      L     L#0;
      U     "MAL1S032Par".Par.FlagProcess.ProcessActive;
      SPBN  n609; // no addition
      SET   ;
      S     "MAL1S032Par".Par.FlagProcess.Inf21; // add heat quantity
      U     "SYS_Scan0_Tick1s"; // scan 1sec
      SPBN  E609;
      L     "MAL1S032Par".Par.ProcessValue_Real.Value05; // heat quantity in kW
      +R    ;
      T     "MAL1S032Par".Par.ProcessValue_Real.Value05;
      SPA   E609;
n609: NOP   0;
      U     "MAL1S032Par".Par.FlagProcess.Inf21; // add heat quantity
      SPBN  E609;
      R     "MAL1S032Par".Par.FlagProcess.Inf21; // add heat quantity
      L     "MAL1S032Par".Par.ProcessValue_Real.Value05;
      L     3.600000e+003;
      /R    ; // from kWs to kWh
      L     1.000000e+003;
      /R    ; // from kWh to MWh
      RND   ;
      T     "MAL1S032Par".Par.ProcessValue_Real.Value06; // result to batch potokoll
      L     0.000000e+000; // clear calculator
      T     "MAL1S032Par".Par.ProcessValue_Real.Value05;
E609: NOP   0;
NETWORK
TITLE =ASW_7000: Step loading kilning
//
      U     "MAL1S032".ToASW.InfDataReady;
      U     "MAL1S032".PCRead.Step.StWait;
      U     "MAL1S032".PCWrite.ExtFuncOn.StartLoading; // PIC command "start loading"
      S     "MAL1S032Par".Par.FlagFunction_1.StepLoading; // Step loading
      R     "MAL1S032Par".Par.FlagMachine.ImpulsNullstellung;
      R     "MAL1S032Par".Par.FlagMachine.CmdTurnRevAfterLoading;
      R     "MAL1S032Par".Par.FlagMachine.CmdTurnFwdAfterLoading;
//
      SET   ;
      R     "MAL1S032".PCWrite.ExtFuncOn.StartLoading; // PIC command "start loading"
//
      U     "MAL1S032".ToASW.InfDataReady;
      U     "MAL1S032".PCRead.Step.StActive;
      U     "MAL1S032Par".Par.FlagFunction_1.StepLoading; // Step loading
      SPB   e71;
      R     "MAL1S032Par".Par.Switches1.StaOn00; // LiftingPositionRound_1
      R     "MAL1S032Par".Par.Switches1.StaOn01; // LiftingPositionRound_2
      R     "MAL1S032Par".Par.Switches1.StaOn02; // LiftingPositionRound_3
      R     "MAL1S032Par".Par.Switches1.StaOn03; // LiftingPositionRound_4
      R     "MAL1S032Par".Par.Switches1.StaOn04; // LiftingPositionRound_5
      R     "MAL1S032Par".Par.Switches1.StaOn05; // LiftingPositionRound_6
e71:  NOP   0;
      U     "MAL1S032".ToASW.InfDataReady;
      U     "MAL1S032".PCRead.Step.StActive;
      U     "MAL1S032Par".Par.FlagFunction_1.StepLoading; // Step loading
      UN    "MAL1S032Par".Par.FlagFunction_1.FinishLoading;
      UN    "MAL1S032Par".Par.FlagFunction_1.LoadEnd;
      SPBN  E700;
      U(    ;
      U(    ;
      L     "G266M".A_3111_MXZ41MA.Ma.OutPositionAngle;
      L     3460; // 346.0°
      >=I   ;
      )     ;
      O     ;
      U(    ;
      L     "G266M".A_3111_MXZ41MA.Ma.OutCntRound;
      L     L#1;
      >=D   ;
      )     ;
      )     ;
      U     "MAL1S032Par".Par.FlagFunction_1.StepLoading;
      =     "MAL1S032Par".Par.FlagFunction_0.ReducedSpeed;
//
      L     "MAL1S032Par".RecipeHeader.Loading.LiftingPositionRound_3;
      L     20; // 20°
      -I    ;
      T     "MAL1S032Par".Par.ParIntMachine.LiftingPositionRound_4;
      L     "MAL1S032Par".RecipeHeader.Loading.LoadingLevelRound_3;
      L     "MAL1S032Par".RecipeHeader.Loading.OffsetLevelNextRound;
      +I    ;
      T     "MAL1S032Par".Par.ParIntMachine.LoadingLevelRound_4;
//
      L     "MAL1S032Par".Par.ParIntMachine.LiftingPositionRound_4;
      L     20; // 20°
      -I    ;
      T     "MAL1S032Par".Par.ParIntMachine.LiftingPositionRound_5;
      L     "MAL1S032Par".Par.ParIntMachine.LoadingLevelRound_4;
      L     "MAL1S032Par".RecipeHeader.Loading.OffsetLevelNextRound;
      +I    ;
      T     "MAL1S032Par".Par.ParIntMachine.LoadingLevelRound_5;
//
      L     "MAL1S032Par".Par.ParIntMachine.LiftingPositionRound_5;
      L     20; // 20°
      -I    ;
      T     "MAL1S032Par".Par.ParIntMachine.LiftingPositionRound_6;
      L     "MAL1S032Par".Par.ParIntMachine.LoadingLevelRound_5;
      L     "MAL1S032Par".RecipeHeader.Loading.OffsetLevelNextRound;
      +I    ;
      T     "MAL1S032Par".Par.ParIntMachine.LoadingLevelRound_6;
//
      L     3600;
      L     "G266M".A_3111_MXZ41MA.Ma.Par.ParTolPosition;
      -I    ;
      L     "G266M".A_3111_MXZ41MA.Ma.OutPositionAngle;
      <=I   ;
      SPB   E700;
//
      L     "G266M".A_3111_MXZ41MA.Ma.OutPositionAngle;
      L     0;
      <I    ;
//      <=I
      SPB   E700;
//
      L     "G266M".A_3111_MXZ41MA.Ma.OutPositionAngle;
      L     10;
      /I    ;
      T     "MAL1S032Par".Par.MachineValue.ISTWERT_FAHRANTRIEB_POSI;
//
      U     "MAL1S032Par".Par.FlagFunction_1.StepLoading; // Step loading
      FP    "MAL1S032Par".Par.Switches1.StaOn08;
      =     "MAL1S032Par".Par.Switches1.StaOn09; // scan start loading
      U     "MAL1S032Par".Par.Switches1.StaOn09; // scan start loading
      SPBN  e72;
      R     "MAL1S032Par".Par.Switches1.StaOn00; // LiftingPositionRound_1
      R     "MAL1S032Par".Par.Switches1.StaOn01; // LiftingPositionRound_2
      R     "MAL1S032Par".Par.Switches1.StaOn02; // LiftingPositionRound_3
      R     "MAL1S032Par".Par.Switches1.StaOn03; // LiftingPositionRound_4
      R     "MAL1S032Par".Par.Switches1.StaOn04; // LiftingPositionRound_5
      R     "MAL1S032Par".Par.Switches1.StaOn05; // LiftingPositionRound_6
//
e72:  NOP   0;
//
      U(    ;
      L     "G266M".A_3111_MXZ41MA.Ma.OutCntRound;
      L     L#0;
      ==D   ;
      )     ;
      U(    ;
      L     "MAL1S032Par".Par.MachineValue.ISTWERT_FAHRANTRIEB_POSI;
      L     "MAL1S032Par".RecipeHeader.Loading.LiftingPositionRound_1;
      <I    ;
      )     ;
      S     "MAL1S032Par".Par.Switches1.StaOn00; // LiftingPositionRound_1
//
      U(    ;
      L     "G266M".A_3111_MXZ41MA.Ma.OutCntRound;
      L     L#0;
      ==D   ;
      )     ;
      U(    ;
      L     "MAL1S032Par".Par.MachineValue.ISTWERT_FAHRANTRIEB_POSI;
      L     "MAL1S032Par".RecipeHeader.Loading.LiftingPositionRound_1;
      >=I   ;
      )     ;
      U(    ;
      L     "MAL1S032Par".Par.MachineValue.ISTWERT_FAHRANTRIEB_POSI;
      L     3550; // 355.0° --> Ruckeln am Nullpunkt abfangen
      <=I   ;
      )     ;
      S     "MAL1S032Par".Par.Switches1.StaOn01; // LiftingPositionRound_2
//
      U     "MAL1S032Par".Par.Switches1.StaOn01; // LiftingPositionRound_2
      R     "MAL1S032Par".Par.Switches1.StaOn00; // LiftingPositionRound_1
//
      U(    ;
      L     "G266M".A_3111_MXZ41MA.Ma.OutCntRound;
      L     L#1;
      ==D   ;
      )     ;
      U(    ;
      L     "MAL1S032Par".Par.MachineValue.ISTWERT_FAHRANTRIEB_POSI;
      L     "MAL1S032Par".RecipeHeader.Loading.LiftingPositionRound_2;
      >=I   ;
      )     ;
      S     "MAL1S032Par".Par.Switches1.StaOn02; // LiftingPositionRound_3
//
      U     "MAL1S032Par".Par.Switches1.StaOn02; // LiftingPositionRound_3
      R     "MAL1S032Par".Par.Switches1.StaOn01; // LiftingPositionRound_2
      R     "MAL1S032Par".Par.Switches1.StaOn00; // LiftingPositionRound_1
//
      U(    ;
      L     "G266M".A_3111_MXZ41MA.Ma.OutCntRound;
      L     L#2;
      ==D   ;
      )     ;
      U(    ;
      L     "MAL1S032Par".Par.MachineValue.ISTWERT_FAHRANTRIEB_POSI;
      L     "MAL1S032Par".RecipeHeader.Loading.LiftingPositionRound_3;
      >=I   ;
      )     ;
      S     "MAL1S032Par".Par.Switches1.StaOn03; // LiftingPositionRound_4
//
      U     "MAL1S032Par".Par.Switches1.StaOn03; // LiftingPositionRound_4
      R     "MAL1S032Par".Par.Switches1.StaOn02; // LiftingPositionRound_3
      R     "MAL1S032Par".Par.Switches1.StaOn01; // LiftingPositionRound_2
      R     "MAL1S032Par".Par.Switches1.StaOn00; // LiftingPositionRound_1
      U(    ;
      L     "G266M".A_3111_MXZ41MA.Ma.OutCntRound;
      L     L#3;
      ==D   ;
      )     ;
      U(    ;
      L     "MAL1S032Par".Par.MachineValue.ISTWERT_FAHRANTRIEB_POSI;
      L     "MAL1S032Par".Par.ParIntMachine.LiftingPositionRound_4;
      >=I   ;
      )     ;
      S     "MAL1S032Par".Par.Switches1.StaOn04; // LiftingPositionRound_5
//
      U     "MAL1S032Par".Par.Switches1.StaOn04; // LiftingPositionRound_5
      R     "MAL1S032Par".Par.Switches1.StaOn03; // LiftingPositionRound_4
      R     "MAL1S032Par".Par.Switches1.StaOn02; // LiftingPositionRound_3
      R     "MAL1S032Par".Par.Switches1.StaOn01; // LiftingPositionRound_2
      R     "MAL1S032Par".Par.Switches1.StaOn00; // LiftingPositionRound_1
      U(    ;
      L     "G266M".A_3111_MXZ41MA.Ma.OutCntRound;
      L     L#4;
      ==D   ;
      )     ;
      U(    ;
      L     "MAL1S032Par".Par.MachineValue.ISTWERT_FAHRANTRIEB_POSI;
      L     "MAL1S032Par".Par.ParIntMachine.LiftingPositionRound_5;
      >=I   ;
      )     ;
      S     "MAL1S032Par".Par.Switches1.StaOn05; // LiftingPositionRound_6
//
      U     "MAL1S032Par".Par.Switches1.StaOn05; // LiftingPositionRound_6
      R     "MAL1S032Par".Par.Switches1.StaOn04; // LiftingPositionRound_5
      R     "MAL1S032Par".Par.Switches1.StaOn03; // LiftingPositionRound_4
      R     "MAL1S032Par".Par.Switches1.StaOn02; // LiftingPositionRound_3
      R     "MAL1S032Par".Par.Switches1.StaOn01; // LiftingPositionRound_2
      R     "MAL1S032Par".Par.Switches1.StaOn00; // LiftingPositionRound_1
      U     "MAL1S032Par".Par.Switches1.StaOn00; // LiftingPositionRound_1
      SPB   Rnd1;
      U     "MAL1S032Par".Par.Switches1.StaOn01; // LiftingPositionRound_2
      SPB   Rnd2;
      U     "MAL1S032Par".Par.Switches1.StaOn02; // LiftingPositionRound_3
      SPB   Rnd3;
      U     "MAL1S032Par".Par.Switches1.StaOn03; // LiftingPositionRound_4
      SPB   Rnd4;
      U     "MAL1S032Par".Par.Switches1.StaOn04; // LiftingPositionRound_5
      SPB   Rnd5;
      U     "MAL1S032Par".Par.Switches1.StaOn05; // LiftingPositionRound_6
      SPB   Rnd6;
      SPA   E700;
Rnd1: NOP   0;
      L     "MAL1S032Par".RecipeHeader.Loading.LoadingLevelRound_1;
      L     "G265M".A_3111_MXZ21_31MA.Ma.Par.ParTolPosition;
      +I    ;
      T     "MAL1S032Par".Par.MachineValue.SOLLWERT_HUBZUG1_HOEHE;
      T     "MAL1S032Par".Par.MachineValue.SOLLWERT_HUBZUG2_HOEHE;
      L     "MAL1S032Par".RecipeHeader.Loading.LoadingSpeed_1;
      T     "MAL1S032Par".Par.MachineValue.SollwertFahrantrieb;
      SPA   E700;
Rnd2: NOP   0;
      L     "MAL1S032Par".RecipeHeader.Loading.LoadingLevelRound_2;
      L     "G265M".A_3111_MXZ21_31MA.Ma.Par.ParTolPosition;
      +I    ;
      T     "MAL1S032Par".Par.MachineValue.SOLLWERT_HUBZUG1_HOEHE;
      T     "MAL1S032Par".Par.MachineValue.SOLLWERT_HUBZUG2_HOEHE;
      L     "MAL1S032Par".RecipeHeader.Loading.LoadingSpeed_2;
      T     "MAL1S032Par".Par.MachineValue.SollwertFahrantrieb;
      SPA   E700;
Rnd3: NOP   0;
      L     "MAL1S032Par".RecipeHeader.Loading.LoadingLevelRound_3;
      L     "G265M".A_3111_MXZ21_31MA.Ma.Par.ParTolPosition;
      +I    ;
      T     "MAL1S032Par".Par.MachineValue.SOLLWERT_HUBZUG1_HOEHE;
      T     "MAL1S032Par".Par.MachineValue.SOLLWERT_HUBZUG2_HOEHE;
      L     "MAL1S032Par".RecipeHeader.Loading.LoadingSpeed_3;
      T     "MAL1S032Par".Par.MachineValue.SollwertFahrantrieb;
      SPA   E700;
Rnd4: NOP   0;
      L     "MAL1S032Par".Par.ParIntMachine.LoadingLevelRound_4;
      L     "G265M".A_3111_MXZ21_31MA.Ma.Par.ParTolPosition;
      +I    ;
      T     "MAL1S032Par".Par.MachineValue.SOLLWERT_HUBZUG1_HOEHE;
      T     "MAL1S032Par".Par.MachineValue.SOLLWERT_HUBZUG2_HOEHE;
//      L     "MAL1S032Par".RecipeHeader.Loading.LoadingSpeed_3
      L     87; // 87%
      T     "MAL1S032Par".Par.MachineValue.SollwertFahrantrieb;
      SPA   E700;
Rnd5: NOP   0;
      L     "MAL1S032Par".Par.ParIntMachine.LoadingLevelRound_5;
      L     "G265M".A_3111_MXZ21_31MA.Ma.Par.ParTolPosition;
      +I    ;
      T     "MAL1S032Par".Par.MachineValue.SOLLWERT_HUBZUG1_HOEHE;
      T     "MAL1S032Par".Par.MachineValue.SOLLWERT_HUBZUG2_HOEHE;
//      L     "MAL1S032Par".RecipeHeader.Loading.LoadingSpeed_3
      L     87; // 87%
      T     "MAL1S032Par".Par.MachineValue.SollwertFahrantrieb;
      SPA   E700;
Rnd6: NOP   0;
      L     "MAL1S032Par".Par.ParIntMachine.LoadingLevelRound_6;
      L     "G265M".A_3111_MXZ21_31MA.Ma.Par.ParTolPosition;
      +I    ;
      T     "MAL1S032Par".Par.MachineValue.SOLLWERT_HUBZUG1_HOEHE;
      T     "MAL1S032Par".Par.MachineValue.SOLLWERT_HUBZUG2_HOEHE;
//      L     "MAL1S032Par".RecipeHeader.Loading.LoadingSpeed_3
      L     87; // 87%
      T     "MAL1S032Par".Par.MachineValue.SollwertFahrantrieb;
      SPA   E700;
E700: NOP   0;
NETWORK
TITLE =Sub 7010: Kilning  loading finished

// Grundschicht vollständig bedeckt
      U(    ;
// Die Position bei IBN ermitteln!
      L     "G266M".A_3111_MXZ41MA.Ma.OutPositionAngle;
      L     3564; // 356.4°
      >=I   ;
      )     ;
      U     "MAL1S032Par".Par.FlagFunction_1.StepLoading;
      U     "G266M".A_3111_MXZ41MA.Ma.InEnableFwd;
      S     "MAL1S032Par".Par.FlagFunction_1.LoadFirstPartEnd;
      S     "MAL1S032Par".Par.FlagProcess.Product_Inside;

      U     "MAL1S032Par".Par.FlagProcess.ProcessActive;
      U     "MAL1S032Par".Par.FlagFunction_1.FinishLoading;
      O     "MAL1S032Par".Par.FlagFunction_1.StepUnloading;
      O     "MAL1S032".PCRead.Step.StIdling; // "SecDB".PCRead.Step.StIdling
      R     "MAL1S032Par".Par.FlagFunction_1.LoadFirstPartEnd;

      L     0;
      L     "MAL1S032".ToSSW.InPrevSecDB;
      ==I   ;
      SPB   fin;
      O(    ;
      U     "MAL1S017Par".Par.FlagFunction_1.FinishUnloading;
      U     "MAL1S017".PCWrite.ExtFuncOn.FinishCleanSurface; // PIC command "finish unloading"
//      U     "MAL1S032".PCWrite.ExtFuncOn.FinishLoading    // PIC command "finish loading"
      O     "MAL1S017Par".Par.FlagFunction_1.StepCleaning;
      U     "MAL1S017".PCRead.Step.StEmptied;
      U(    ;
      AUF   "MAL1S017";
      L     DBNO;
      L     "MAL1S032".ToSSW.InPrevSecDB;
      ==I   ;
      )     ;
      )     ;
      O(    ;
      U     "MAL1S018Par".Par.FlagFunction_1.FinishUnloading;
      U     "MAL1S018".PCWrite.ExtFuncOn.FinishCleanSurface; // PIC command "finish unloading"
//      U     "MAL1S032".PCWrite.ExtFuncOn.FinishLoading    // PIC command "finish loading"
      O     "MAL1S018Par".Par.FlagFunction_1.StepCleaning;
      U     "MAL1S018".PCRead.Step.StEmptied;
      U(    ;
      AUF   "MAL1S018";
      L     DBNO;
      L     "MAL1S032".ToSSW.InPrevSecDB;
      ==I   ;
      )     ;
      )     ;
      O(    ;
      U     "MAL1S019Par".Par.FlagFunction_1.FinishUnloading;
      U     "MAL1S019".PCWrite.ExtFuncOn.FinishCleanSurface; // PIC command "finish unloading"
//      U     "MAL1S032".PCWrite.ExtFuncOn.FinishLoading    // PIC command "finish loading"
      O     "MAL1S019Par".Par.FlagFunction_1.StepCleaning;
      U     "MAL1S019".PCRead.Step.StEmptied;
      U(    ;
      AUF   "MAL1S019";
      L     DBNO;
      L     "MAL1S032".ToSSW.InPrevSecDB;
      ==I   ;
      )     ;
      )     ;
      O(    ;
      U     "MAL1S020Par".Par.FlagFunction_1.FinishUnloading;
      U     "MAL1S020".PCWrite.ExtFuncOn.FinishCleanSurface; // PIC command "finish unloading"
//      U     "MAL1S032".PCWrite.ExtFuncOn.FinishLoading    // PIC command "finish loading"
      O     "MAL1S020Par".Par.FlagFunction_1.StepCleaning;
      U     "MAL1S020".PCRead.Step.StEmptied;
      U(    ;
      AUF   "MAL1S020";
      L     DBNO;
      L     "MAL1S032".ToSSW.InPrevSecDB;
      ==I   ;
      )     ;
      )     ;
      O(    ;
      U     "MAL1S021Par".Par.FlagFunction_1.FinishUnloading;
      U     "MAL1S021".PCWrite.ExtFuncOn.FinishCleanSurface; // PIC command "finish unloading"
//      U     "MAL1S032".PCWrite.ExtFuncOn.FinishLoading    // PIC command "finish loading"
      O     "MAL1S021Par".Par.FlagFunction_1.StepCleaning;
      U     "MAL1S021".PCRead.Step.StEmptied;
      U(    ;
      AUF   "MAL1S021";
      L     DBNO;
      L     "MAL1S032".ToSSW.InPrevSecDB;
      ==I   ;
      )     ;
      )     ;
      O(    ;
      U     "MAL1S022Par".Par.FlagFunction_1.FinishUnloading;
      U     "MAL1S022".PCWrite.ExtFuncOn.FinishCleanSurface; // PIC command "finish unloading"
//      U     "MAL1S032".PCWrite.ExtFuncOn.FinishLoading    // PIC command "finish loading"
      O     "MAL1S022Par".Par.FlagFunction_1.StepCleaning;
      U     "MAL1S022".PCRead.Step.StEmptied;
      U(    ;
      AUF   "MAL1S022";
      L     DBNO;
      L     "MAL1S032".ToSSW.InPrevSecDB;
      ==I   ;
      )     ;
      )     ;
      O(    ;
      U     "MAL1S023Par".Par.FlagFunction_1.FinishUnloading;
      U     "MAL1S023".PCWrite.ExtFuncOn.FinishCleanSurface; // PIC command "finish unloading"
//      U     "MAL1S032".PCWrite.ExtFuncOn.FinishLoading    // PIC command "finish loading"
      O     "MAL1S032Par".Par.FlagFunction_1.StepCleaning;
      U     "MAL1S032".PCRead.Step.StEmptied;
      U(    ;
      AUF   "MAL1S023";
      L     DBNO;
      L     "MAL1S023".ToSSW.InPrevSecDB;
      ==I   ;
      )     ;
      )     ;
      O(    ;
      U     "MAL1S024Par".Par.FlagFunction_1.FinishUnloading;
      U     "MAL1S024".PCWrite.ExtFuncOn.FinishCleanSurface; // PIC command "finish unloading"
//      U     "MAL1S032".PCWrite.ExtFuncOn.FinishLoading    // PIC command "finish loading"
      O     "MAL1S024Par".Par.FlagFunction_1.StepCleaning;
      U     "MAL1S024".PCRead.Step.StEmptied;
      U(    ;
      AUF   "MAL1S024";
      L     DBNO;
      L     "MAL1S032".ToSSW.InPrevSecDB;
      ==I   ;
      )     ;
      )     ;
//      O(
//      U     "MAL1S032Par".Par.FlagFunction_1.StepLoading    // Step loading
//      UN    "MAL1S032".ToASW.InfSameJobPrevSec
//      U     "MAL1S032".PCWrite.ExtFuncOn.FinishLoading    // PIC command "finish loading"
//      )
      U     "MAL1S032".ToASW.InfDataReady;
      U     "MAL1S032".PCRead.Step.StActive;
      U     "MAL1S032Par".Par.FlagFunction_1.LoadFirstPartEnd;
      S     "MAL1S032Par".Par.FlagFunction_1.LoadEnd;
      R     "MAL1S017".PCWrite.ExtFuncOn.FinishCleanSurface; // PIC command "finish unloading"
      R     "MAL1S018".PCWrite.ExtFuncOn.FinishCleanSurface; // PIC command "finish unloading"
      R     "MAL1S019".PCWrite.ExtFuncOn.FinishCleanSurface; // PIC command "finish unloading"
      R     "MAL1S020".PCWrite.ExtFuncOn.FinishCleanSurface; // PIC command "finish unloading"
      R     "MAL1S021".PCWrite.ExtFuncOn.FinishCleanSurface; // PIC command "finish unloading"
      R     "MAL1S022".PCWrite.ExtFuncOn.FinishCleanSurface; // PIC command "finish unloading"
      R     "MAL1S023".PCWrite.ExtFuncOn.FinishCleanSurface; // PIC command "finish unloading"
      R     "MAL1S024".PCWrite.ExtFuncOn.FinishCleanSurface; // PIC command "finish unloading"

//
      U     "MAL1S032".PCWrite.ExtFuncOn.FinishLoading; // PIC command "finish loading"
      R     "MAL1S032".PCWrite.ExtFuncOn.FinishLoading; // PIC command "finish loading"
//
      U     "MAL1S032Par".Par.FlagFunction_1.LoadEnd;
      U     "MAL1S032Par".Par.FlagFunction_1.StepLoading; // Step loading
      FP    "MAL1S032Par".Par.FlagFunction_0.ImpulsSollposition;
      =     "MAL1S032Par".Par.FlagFunction_0.MerkerSollpositionFP;
      U     "MAL1S032Par".Par.FlagFunction_0.MerkerSollpositionFP;
      SPBN  fin;
      L     "G266M".A_3111_MXZ41MA.Ma.OutPositionAngle;
      L     "MAL1S032Par".Par.ParIntProcess.LoadingOverlap;
      +I    ;
      T     "G266M".A_3111_MXZ41MA.Ma.InPositionTarget;
      SET   ;
      S     "G266M".TurningTo_Parkposition;

// Extra Planierrunde wenn der Fahrantrieb ueber 346° beim Beladen Ende war
      L     "G266M".A_3111_MXZ41MA.Ma.OutPositionAngle;
      L     3460; // 346,0 °
      >I    ;
      S     "G266M".Turning_One_Round_More;

// Beladehöhe speichern
      L     "MAL1S032Par".Par.MachineValue.SOLLWERT_HUBZUG1_HOEHE;
      T     "MAL1S032Par".Par.ParIntMachine.LastLoadingLevel; // saved loading value
fin:  NOP   0;

// Hubzüge erst auf der Parkposition abheben
      U     "G266M".TurningTo_Parkposition;
      FN    "G265M".USW8;
      =     "G265M".USW9;

      U     "G265M".USW9;
      O     ;
      U     "MAL1S032Par".Par.FlagFunction_1.FinishLoading;
      U(    ;
      U     "G266M".A_3111_MXZ41MA.A_3111_BZS43.StCtoTrue; // sensor zero point
      O     "G266M".A_3111_MXZ41MA.A_3111_BZS43.StTrue; // sensor zero point
      )     ;
      SPBN  auf;
      L     "G265M".A_3111_MXZ21_31MA.Ma.Par.ParPositionTopLeftUnits; //LIFTING DRIVE
      L     150;
      +I    ;
      T     "MAL1S032Par".Par.MachineValue.SOLLWERT_HUBZUG1_HOEHE;
      L     "G265M".A_3111_MXZ21_31MA.Ma.Par.ParPositionTopRightUnits; //LIFTING DRIVE
      L     150;
      +I    ;
      T     "MAL1S032Par".Par.MachineValue.SOLLWERT_HUBZUG2_HOEHE;
      L     1;
      T     "G265M".A_3111_MXZ21_31MA.Ma.Par.ParTolPosition;
auf:  NOP   0;

      NOP   0;
NETWORK
TITLE =ASW_6080: Processtime Kilning
//      CALL  "SSA_MH_ProcessTime_Fct" , DB1017
//       InfDataReady :="MAL1S017".ToASW.InfDataReady
//       ProzessActive:="MAL1S017Par".Par.FlagProcess.ProcessActive
//       InStartTime  :="MAL1S017Par".Prozesstime.Starttime
//       OutStartTime :="MAL1S017Par".Prozesstime.Starttime
//       ProcessTime  :="MAL1S017Par".Prozesstime
//
      CALL "SSA_MH_ProcessTime_Fct" , DB  1032 (
           InfDataReady             := "MAL1S032".ToASW.InfDataReady,
           ProzessActive            := "MAL1S032Par".Par.FlagProcess.ProcessActive,
           InStartTime              := "MAL1S032Par".Processtime.StartTime,
           OutStartTime             := "MAL1S032Par".Processtime.StartTime,
           ProcessTime              := "MAL1S032Par".Processtime);

NETWORK
TITLE =Sub 7020: Step start process kilning

      U     "MAL1S032".ToASW.InfDataReady;
      U     "MAL1S032".PCRead.Step.StActive;
//      U     "MAL1S032".PCWrite.ExtFuncOn.StartProcess    // PIC command "start process kilning"
      U     "MAL1S032Par".Par.FlagFunction_1.LoadEnd;

      U     "G266M".A_3111_MXZ41MA.A_3111_BZS43.StTrue; // sensor zero point
      U     "G265M".A_3111_MXZ21_31MA.A_3111_BZS23.InpTrue;
      U     "G265M".A_3111_MXZ21_31MA.A_3111_BZS33.InpTrue;

      O(    ;
      UN    "MAL1S032".SecNom.Par1On.Cmd01; // With Loading
      UN    "MAL1S032".ToASW.InfSameBatchPrevSec;
      U     "MAL1S032".ToASW.InfDataReady;
      U     "MAL1S032".PCRead.Step.StActive;
      )     ;

      S     "MAL1S032Par".Par.FlagFunction_1.FinishLoading; // start process kilning
      R     "MAL1S032Par".Par.FlagFunction_1.LoadEnd;
//
      U     "MAL1S032".PCWrite.ExtFuncOn.StartProcess; // PIC command "start process kilning"
      R     "MAL1S032".PCWrite.ExtFuncOn.StartProcess; // PIC command "start process kilning"
//
      U     "G266M".A_3111_MXZ41MA.Ma.StAdjusted;
      O     "G266M".A_3111_MXZ41MA.Ma.OutAdjusted;
      U     "MAL1S032Par".Par.FlagFunction_1.FinishLoading; // start process kilning
      O     "MAL1S032Par".Par.FlagProcess.ProcessActive;
      SPBN  E702;
      L     "G265M".A_3111_MXZ21_31MA.Ma.Par.ParPositionTopLeftUnits; //LIFTING DRIVE
      L     50; //jk
      +I    ;
      T     "MAL1S032Par".Par.MachineValue.SOLLWERT_HUBZUG1_HOEHE;
      L     "G265M".A_3111_MXZ21_31MA.Ma.Par.ParPositionTopRightUnits; //LIFTING DRIVE
      L     50; //jk
      +I    ;
      T     "MAL1S032Par".Par.MachineValue.SOLLWERT_HUBZUG2_HOEHE;
      L     1;
      T     "G265M".A_3111_MXZ21_31MA.Ma.Par.ParTolPosition;

E702: NOP   0;

      U     "G266M".TurningTo_Parkposition;
      SPBN  E703;
      U(    ;
      L     "G266M".A_3111_MXZ41MA.Ma.OutPositionAngle;
      L     3500;
      >=I   ;
      )     ;
      SPBN  E703;
      L     10; // 10% speed to parkposition
      T     "MAL1S032Par".Par.MachineValue.SollwertFahrantrieb;
E703: NOP   0;

      U     "G266M".TurningTo_Parkposition;
      SPBN  E704;
      U(    ;
      L     "G266M".A_3111_MXZ41MA.Ma.OutPositionAngle;
      L     3500;
      <I    ;
      )     ;
      SPBN  E704;
      L     87; // 87% speed to parkposition
      T     "MAL1S032Par".Par.MachineValue.SollwertFahrantrieb;
E704: NOP   0;

NETWORK
TITLE =ASW_8000:  Step unloading kilning

      UN    "MAL1S032Par".Par.FlagFunction_1.StepUnloading; // Step Unloading
      R     "MAL1S032Par".Par.FlagFunction_0.OverlapSaved; // Ueberlappung erfasst
//
      U     "MAL1S032".ToASW.InfDataReady;
      U     "MAL1S032".PCRead.Step.StEmptying;
      U(    ;
      L     "MAL1S032Par".RecipeHeader.Unloading.StartUnloadAuto; //StartUnloadAuto = 0
      L     1;
      <>I   ;
      U     "MAL1S032".PCWrite.ExtFuncOn.StartUnLoading; // PIC command "start unloading"
      O     ;
      U(    ;
      L     "MAL1S032Par".RecipeHeader.Unloading.StartUnloadAuto; //StartUnloadAuto = 10
      L     1;
      ==I   ;
      )     ;
      UN    DB371.DBX  832.1; // 30% Ventilatordrehzahl
      UN    DB371.DBX 1856.1; // 30% Ventilatordrehzahl
      )     ;
      S     "MAL1S032Par".Par.FlagFunction_1.StepUnloading; // Step Unloading
      R     "MAL1S032Par".Par.FlagMachine.ImpulsNullstellung;
      R     "MAL1S023Par".Par.FlagMachine.WEGMESSUNG_0;
      R     DB922.DBX  148.0; // FP
      R     "MAL1S032Par".Par.FlagMachine.CmdTurnRevAfterUnloading;
      R     "MAL1S032Par".Par.FlagMachine.CmdTurnFwdAfterUnloading;
//
      SET   ;
      R     "MAL1S032".PCWrite.ExtFuncOn.StartUnLoading; // PIC command "start unloading"
//
      U     "MAL1S032".ToASW.InfDataReady;
      U     "MAL1S032".PCRead.Step.StEmptying;
      U     "MAL1S032Par".Par.FlagFunction_1.StepUnloading; // Step Unloading
      SPBN  e800;
      L     "MAL1S032Par".Par.ParIntMachine.LastLoadingLevel; // saved loading value
      T     "MAL1S032Par".Par.ParIntMachine.FUELLHOEHE_PRODUKT;
//
      U(    ;
      L     "G265M".A_3111_MXZ21_31MA.Ma.OutPositionLeft;
      L     "MAL1S032Par".Par.ParIntMachine.FUELLHOEHE_PRODUKT;
      >I    ;
      )     ;
      O(    ;
      L     "G265M".A_3111_MXZ21_31MA.Ma.OutPositionRight;
      L     "MAL1S032Par".Par.ParIntMachine.FUELLHOEHE_PRODUKT;
      >I    ;
      )     ;
      UN(   ;
      U(    ;
      L     "G265M".A_3111_MXZ21_31MA.Ma.OutPositionLeft;
      L     "MAL1S032Par".Par.MachineValue.SOLLWERT_HUBZUG1_HOEHE;
      <=I   ;
      )     ;
      U(    ;
      L     "G265M".A_3111_MXZ21_31MA.Ma.OutPositionRight;
      L     "MAL1S032Par".Par.MachineValue.SOLLWERT_HUBZUG1_HOEHE;
      <=I   ;
      )     ;
      )     ;
      =     "MAL1S032Par".Par.FlagFunction_0.ScrewAboveProductLayer; // HubzuegeUeberProdukt
//
//- Letzte Entladehoehe erreicht ---
      U(    ;
      L     "MAL1S032Par".Par.MachineValue.SOLLWERT_HUBZUG1_HOEHE;
      L     0;
      <=I   ;
      )     ;
      U(    ;
      L     "MAL1S032Par".Par.MachineValue.SOLLWERT_HUBZUG1_HOEHE;
      L     "G265M".A_3111_MXZ21_31MA.Ma.InPositionTarget;
      ==I   ;
      )     ;
      U     "G265M".A_3111_MXZ21_31MA.Ma.StAdjusted;
      U     "MAL1S032Par".Par.FlagFunction_1.StepUnloading; // Step Unloading
      FP    "MAL1S032Par".Par.FlagFunction_0.UnloadLevelReachedFP; // UnloadLevelReachedFP
      =     "MAL1S032Par".Par.FlagFunction_0.ImpulsUnloadLevelReached; // ImpulsUnloadLevelReached
      UN    "MAL1S032Par".Par.FlagFunction_0.ImpulsUnloadLevelReached; // ImpulsUnloadLevelReached
      O     "MAL1S032Par".Par.FlagFunction_0.OverlapSaved; // Ueberlappung erfasst
      SPB   over;
      L     "G266M".A_3111_MXZ41MA.Ma.OutCntRound;
      L     1;
      +I    ;
      T     "MAL1S032Par".Par.ParIntProcess.UnloadungRounds;
//
      L     "G266M".A_3111_MXZ41MA.Ma.OutPositionAngle;
      L     3600; // 360,0°
      >=I   ;
      SPBN  soz1;
      -I    ;
      SPA   soz2;
soz1: NOP   0;
      TAK   ;
soz2: NOP   0;
      L     100; // 10,0°
      +I    ;
      T     "MAL1S032Par".Par.ParIntProcess.UnloadingOverlap;
      T     "G266M".A_3111_MXZ41MA.Ma.InPositionTarget;
      S     "MAL1S032Par".Par.FlagFunction_0.OverlapSaved; // Ueberlappung erfasst
over: NOP   0;
      U(    ;
      L     "G266M".A_3111_MXZ41MA.Ma.OutCntRound;
      L     L#0;
      ==D   ;
      )     ;
      SPB   rnd1;
      L     "G266M".A_3111_MXZ41MA.Ma.OutCntRound;
      L     L#1;
      ==D   ;
      SPB   rnd2;
      L     "G266M".A_3111_MXZ41MA.Ma.OutCntRound;
      L     L#2;
      >=D   ;
      SPB   rnd3;
      SPA   e801;
rnd1: NOP   0;
      L     "MAL1S032Par".RecipeHeader.Unloading.UnLoadingLevelRound_1;
      T     "MAL1S032Par".Par.MachineValue.SOLLWERT_HUBZUG1_HOEHE;
      T     "MAL1S032Par".Par.MachineValue.SOLLWERT_HUBZUG2_HOEHE;
      L     1;
      T     "G265M".A_3111_MXZ21_31MA.Ma.Par.ParTolPosition;
      L     "MAL1S032Par".RecipeHeader.Unloading.UnLoadingSpeed_1;
      T     "MAL1S032Par".Par.MachineValue.SollwertFahrantrieb;
      SPA   e801;
rnd2: NOP   0;
      L     "MAL1S032Par".RecipeHeader.Unloading.UnLoadingLevelRound_2;
      T     "MAL1S032Par".Par.MachineValue.SOLLWERT_HUBZUG1_HOEHE;
      T     "MAL1S032Par".Par.MachineValue.SOLLWERT_HUBZUG2_HOEHE;
      L     1;
      T     "G265M".A_3111_MXZ21_31MA.Ma.Par.ParTolPosition;
      L     "MAL1S032Par".RecipeHeader.Unloading.UnLoadingSpeed_2;
      T     "MAL1S032Par".Par.MachineValue.SollwertFahrantrieb;
      SPA   e801;
rnd3: NOP   0;
      L     "MAL1S032Par".RecipeHeader.Unloading.UnLoadingLevelRound_3;
      T     "MAL1S032Par".Par.MachineValue.SOLLWERT_HUBZUG1_HOEHE;
      T     "MAL1S032Par".Par.MachineValue.SOLLWERT_HUBZUG2_HOEHE;
      L     1;
      T     "G265M".A_3111_MXZ21_31MA.Ma.Par.ParTolPosition;
      L     "MAL1S032Par".RecipeHeader.Unloading.UnLoadingSpeed_3;
      T     "MAL1S032Par".Par.MachineValue.SollwertFahrantrieb;
      SPA   e801;

e801: NOP   0;
      U     "MAL1S032".ToASW.InfDataReady;
      U     "MAL1S032".PCRead.Step.StEmptying;
      U     "MAL1S032Par".Par.FlagFunction_1.StepUnloading; // Step Unloading
      U(    ;
      L     "G266M".A_3111_MXZ41MA.Ma.OutCntRound;
      L     "MAL1S032Par".Par.ParIntProcess.UnloadungRounds;
      >=I   ;
      )     ;
      U     "G265M".A_3111_MXZ21_31MA.Ma.StAdjusted;
      U     "G266M".A_3111_MXZ41MA.Ma.StAdjusted;
      S     "MAL1S032Par".Par.FlagFunction_1.FinishUnloading;

      U     "MAL1S032".ToASW.InfDataReady;
      U     "MAL1S032".PCRead.Step.StEmptying;
      U     "MAL1S032Par".Par.FlagFunction_1.FinishUnloading;
      SPBN  e800;
      L     "G265M".A_3111_MXZ21_31MA.Ma.Par.ParPositionTopLeftUnits;
      L     50;
      +I    ;
      T     "MAL1S032Par".Par.MachineValue.SOLLWERT_HUBZUG1_HOEHE;
      L     "G265M".A_3111_MXZ21_31MA.Ma.Par.ParPositionTopRightUnits;
      L     50;
      +I    ;
      T     "MAL1S032Par".Par.MachineValue.SOLLWERT_HUBZUG2_HOEHE;
      L     1;
      T     "G265M".A_3111_MXZ21_31MA.Ma.Par.ParTolPosition;

      L     0;
      T     "MAL1S032Par".Par.ParIntMachine.LastLoadingLevel; // saved loading value
      T     "MAL1S032Par".Par.ParIntMachine.FUELLHOEHE_PRODUKT;
e800: NOP   0;
//
// --> Wie bei der Bank Avangard
      U     "MAL1S032Par".Par.FlagFunction_1.StepUnloading;
      U     "MAL1S032Par".Par.FlagFunction_1.FinishUnloading;
      FP    DB922.DBX  148.0;
      =     DB922.DBX  148.1;
      SPBN  TAU1;
      L     "G266M".A_3111_MXZ41MA.Ma.OutPositionAngle;
      L     1800;
      <I    ;
      S     "MAL1S032Par".Par.FlagMachine.CmdTurnRevAfterUnloading;
      L     "G266M".A_3111_MXZ41MA.Ma.OutPositionAngle;
      L     1800;
      >=I   ;
      S     "MAL1S032Par".Par.FlagMachine.CmdTurnFwdAfterUnloading;
TAU1: NOP   0;
      U     "MAL1S032Par".Par.FlagMachine.CmdTurnRevAfterUnloading;
      O     "MAL1S032Par".Par.FlagMachine.CmdTurnFwdAfterUnloading;
      U     "MAL1S032Par".Par.FlagFunction_1.FinishUnloading;
      U     "G267M".A_3111_MXZ11.StStopped;
      U     "G265M".A_3111_MXZ21_31MA.Ma.OutHigherMinPos;
      U(    ;
      U     "G265M".A_3111_MXZ21_31MA.A_3111_BZS33.InpTrue;
      U     "G265M".A_3111_MXZ21_31MA.A_3111_BZS23.InpTrue;
      O     "G265M".A_3111_MXZ21_31MA.Ma.StAdjusted;
      )     ;
      S     "MAL1S032Par".Par.FlagMachine.WEGMESSUNG_0;
//
      U     "MAL1S032".ToASW.InfDataReady;
      U     "MAL1S032Par".Par.FlagFunction_1.FinishUnloading;
      U     "MAL1S032Par".Par.FlagMachine.WEGMESSUNG_0;
      SPBN  TAU2;
//    L     "MAL1S032Par".RecipeHeader.Cleaning.CleaningSpeed_1
      L     30; // 30%
      T     "MAL1S032Par".Par.MachineValue.SollwertFahrantrieb;
TAU2: NOP   0;
      NOP   0;
NETWORK
TITLE =ASW_9000: Step cleaning
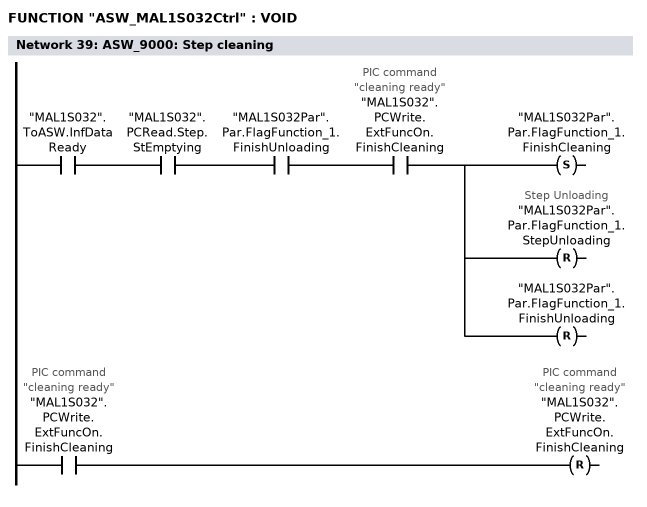

      U     "MAL1S032".ToASW.InfDataReady;
      U     "MAL1S032".PCRead.Step.StEmptying;
      U     "MAL1S032Par".Par.FlagFunction_1.FinishUnloading;
      U     "MAL1S032".PCWrite.ExtFuncOn.FinishCleaning; // PIC command "cleaning ready"
      S     "MAL1S032Par".Par.FlagFunction_1.FinishCleaning;
      R     "MAL1S032Par".Par.FlagFunction_1.StepUnloading; // Step Unloading
      R     "MAL1S032Par".Par.FlagFunction_1.FinishUnloading;
//
      U     "MAL1S032".PCWrite.ExtFuncOn.FinishCleaning; // PIC command "cleaning ready"
      R     "MAL1S032".PCWrite.ExtFuncOn.FinishCleaning; // PIC command "cleaning ready"
NETWORK
TITLE =ASW_9080: Send section date to PIC after germination

      AUF   "MAL1S032";
      U     "MAL1S032".PCRead.Step.StEmptying;
      FP    "MAL1S032Par".Par.FlagProcess.FP_SendResultToPIC;
      SPBN  E908;
//

E908: NOP   0;
NETWORK
TITLE =ASW_10000: ILO functions

      U     "MAL1S032".SecAc.Sta1On.Inf08;
      =     "MAL1S032".Gr.All.Spare04;

//- Little help for PIC-People, Number 3
      UN    "G265M".Gr.InManual; // LIFTING DEVICE KILN 1
      UN    "G266M".Gr.InManual; // TRAVELLING DRIVE KILN 1
      UN    "G267M".Gr.InManual; // UNLOADING / LOADING SCREW KILN 1
      UN    "G268M".Gr.InManual; // DISCHARGE DOOR KILN 1
      UN    "G271M".Gr.InManual; // FAN KILN 1
      UN    "G272M".Gr.InManual; // FRESH AIR LOUVER KILN 1
      UN    "G273M".Gr.InManual; // RECYCLING AIR LOUVER KILN 1
      UN    "G274M".Gr.InManual; // EXHAUST AIR LOUVER KILN 1
      UN    "G276M".Gr.InManual; // HEATING KILN 1
      UN    "G277M".Gr.InManual; // LOUVER AIR HEATER 1 FOR KILN 1
      UN    "G278M".Gr.InManual; // WITHERING AIR KILN 1
      UN    "G279M".Gr.InManual; // HEATING KILN 1 + 2
      FP    DB922.DBX 3029.0;
      =     DB922.DBX 3029.1;
      U     DB922.DBX 3029.1;
      SPBN  RSM3;
      L     0;
      T     "MAL1S032Par".Ilo.Code_ILO_Funktion0; // FCM 32 LINE 1 SEC 32 KILN
      T     "MAL1S032Par".Ilo.ILOMode;
RSM3: NOP   0;

//- Combination OLD and NEW ---
      U     "MAL1S032".SecAc.Sta1On.Inf08;
      SPBN  IFM;
      L     "MAL1S032Par".Ilo.ILOMode;
      L     100;
      *I    ;
      T     "MAL1S032Par".Ilo.Code_ILO_Funktion0;
IFM:  NOP   0;

//  no ILO-mode >> cmd manual off to all used groups and reset all flags
      U     "MAL1S032".SecAc.Sta1On.Inf08;
      FN    "MAL1S032Par".Ilo.Flag.EdgeILOModeOn;
      S     "MAL1S032Par".Ilo.GrCMDManOff[1]; // (ManOff)
      R     "MAL1S032Par".Ilo.GrCMDManAdditional.Cmd1[1];
      R     "MAL1S032Par".Ilo.GrCMDManAdditional.Cmd2[2];
//  Gr-cmd manual OFF
      S     "G265M".Gr.CmdManualOff; // LIFTING DEVICE KILN 1
      S     "G266M".Gr.CmdManualOff; // TRAVELLING DRIVE KILN 1
      S     "G267M".Gr.CmdManualOff; // UNLOADING / LOADING SCREW KILN 1
      S     "G268M".Gr.CmdManualOff; // DISCHARGE DOOR KILN 1
      S     "G271M".Gr.CmdManualOff; // FAN KILN 1
      S     "G272M".Gr.CmdManualOff; // FRESH AIR LOUVER KILN 1
      S     "G273M".Gr.CmdManualOff; // RECYCLING AIR LOUVER KILN 1
      S     "G274M".Gr.CmdManualOff; // EXHAUST AIR LOUVER KILN 1
      S     "G276M".Gr.CmdManualOff; // HEATING KILN 1
      S     "G277M".Gr.CmdManualOff; // LOUVER AIR HEATER 1 FOR KILN 1
      S     "G278M".Gr.CmdManualOff; // WITHERING AIR KILN 1
      S     "G279M".Gr.CmdManualOff; // HEATING KILN 1 + 2
//  RESET ADDITIONAL CMD`S
      R     "G265M".USW14; // ILO-cmd
      R     "G265M".USW15; // ILO-cmd
      R     "G266M".USW14; // ILO-cmd
      R     "G266M".USW15; // ILO-cmd
      R     "G267M".USW14; // ILO-cmd
      R     "G267M".USW15; // ILO-cmd
      R     "G268M".USW14; // ILO-cmd
      R     "G268M".USW15; // ILO-cmd
      R     "G271M".USW14; // ILO-cmd
      R     "G271M".USW15; // ILO-cmd
      R     "G272M".USW14; // ILO-cmd
      R     "G272M".USW15; // ILO-cmd
      R     "G273M".USW14; // ILO-cmd
      R     "G273M".USW15; // ILO-cmd
      R     "G274M".USW14; // ILO-cmd
      R     "G274M".USW15; // ILO-cmd
      R     "G276M".USW14; // ILO-cmd
      R     "G276M".USW15; // ILO-cmd
      R     "G277M".USW14; // ILO-cmd
      R     "G277M".USW15; // ILO-cmd
      R     "G278M".USW14; // ILO-cmd
      R     "G278M".USW15; // ILO-cmd
      R     "G279M".USW14; // ILO-cmd
      R     "G279M".USW15; // ILO-cmd

      NOP   0;
// --- FCM 01 - Lifting devices ---
      L     "MAL1S032Par".Ilo.ILOMode;
      L     1;
      <>I   ;
      SPB   IO1;
// man on
      U     "MAL1S032Par".Ilo.GrCMDManOn[1];
      S     "G265M".Gr.InManual; // LIFTING DEVICE KILN 1
      R     "MAL1S032Par".Ilo.GrCMDManOn[1];
// man off
      U     "MAL1S032Par".Ilo.GrCMDManOff[1];
      S     "G265M".Gr.CmdManualOff; // LIFTING DEVICE KILN 1
      R     "G265M".Gr.InManual; // LIFTING DEVICE KILN 1
      R     "G265M".USW14; // ILO-cmd
      R     "G265M".USW15; // ILO-cmd
      R     "MAL1S032Par".Ilo.GrCMDManOff[1];
      R     "MAL1S032Par".Ilo.GrCMDManAdditional.Cmd1[1];
      R     "MAL1S032Par".Ilo.GrCMDManAdditional.Cmd2[1];
// man start
      U     "MAL1S032Par".Ilo.GrCMDManStart[1];
      S     "G265M".Gr.CmdOn; // LIFTING DEVICE KILN 1
      S     "G265M".Gr.CmdContinue; // LIFTING DEVICE KILN 1
      R     "MAL1S032Par".Ilo.GrCMDManStart[1];
      U     "MAL1S032Par".Ilo.GrCMDManStart[2];
      R     "MAL1S032Par".Ilo.GrCMDManStart[2];
// man stop
      U     "MAL1S032Par".Ilo.GrCMDManStop[1];
      S     "G265M".Gr.CmdOff; // LIFTING DEVICE KILN 1
      R     "MAL1S032Par".Ilo.GrCMDManStop[1];
// man fault reset
      U     "MAL1S032Par".Ilo.GrCMDManFaultReset[1];
      S     "G265M".Gr.CmdFaultReset; // LIFTING DEVICE KILN 1
      R     "MAL1S032Par".Ilo.GrCMDManFaultReset[1];
// moving direction
      UN    "G265M".Gr.InManual; // LIFTING DEVICE KILN 1
      O(    ;
      L     "MAL1S032Par".Ilo.Code_ILO_Funktion0;
      L     100;
      <>I   ;
      )     ;
      SPB   Stat;
      UN    "MAL1S032Par".Ilo.GrCMDManAdditional.Cmd1[1];
      UN    "MAL1S032Par".Ilo.GrCMDManAdditional.Cmd2[1];
      L     "MAL1S032Par".Par.MachineValue.SOLLWERT_HUBZUG1_HOEHE;
      SPB   Tpos;
      U     "MAL1S032Par".Ilo.GrCMDManAdditional.Cmd1[1]; // ManUp
      L     2000; // 1850mm + Offset = 2000mm
      SPB   Tpos;
      U     "MAL1S032Par".Ilo.GrCMDManAdditional.Cmd2[1]; // ManDown
      L     0; // 0mm
      SPB   Tpos;
      SPA   Stat;
// target position
Tpos: NOP   0;
      T     "MAL1S032Par".Par.ParIntProcess.TarPos_ILO_LiftDev;
Stat: NOP   0;
IO1:  NOP   0;
      NOP   0;
// --- FCM 04 - Fans ---
      L     "MAL1S032Par".Ilo.ILOMode;
      L     4;
      <>I   ;
      SPB   IO4;
// man on
      U     "MAL1S032Par".Ilo.GrCMDManOn[1];
      S     "G271M".Gr.InManual; // FAN KILN 1
      R     "MAL1S032Par".Ilo.GrCMDManOn[1];
// man off
      U     "MAL1S032Par".Ilo.GrCMDManOff[1];
      S     "G271M".Gr.CmdManualOff; // FAN KILN 1
      R     "G271M".Gr.InManual; // FAN KILN 1
      R     "G271M".USW14; // ILO-cmd
      R     "G271M".USW15; // ILO-cmd
      R     "MAL1S032Par".Ilo.GrCMDManOff[1];
      R     "MAL1S032Par".Ilo.GrCMDManAdditional.Cmd1[1];
      R     "MAL1S032Par".Ilo.GrCMDManAdditional.Cmd2[1];
// man start
      U     "MAL1S032Par".Ilo.GrCMDManStart[1];
      S     "G271M".Gr.CmdOn; // FAN KILN 1
      S     "G271M".Gr.CmdContinue; // FAN KILN 1
      R     "MAL1S032Par".Ilo.GrCMDManStart[1];
      U     "MAL1S032Par".Ilo.GrCMDManStart[2];
      R     "MAL1S032Par".Ilo.GrCMDManStart[2];
// man stop
      U     "MAL1S032Par".Ilo.GrCMDManStop[1];
      S     "G271M".Gr.CmdOff; // FAN KILN 1
      R     "MAL1S032Par".Ilo.GrCMDManStop[1];
// man fault reset
      U     "MAL1S032Par".Ilo.GrCMDManFaultReset[1];
      S     "G271M".Gr.CmdFaultReset; // FAN KILN 1
      R     "MAL1S032Par".Ilo.GrCMDManFaultReset[1];
// target position
      UN    "G271M".Gr.InManual; // FAN KILN 1
      O(    ;
      L     "MAL1S032Par".Ilo.Code_ILO_Funktion0;
      L     400;
      <>I   ;
      )     ;
      SPB   F04a;
      L     "MAL1S032Par".Ilo.SetpointInt01[1];
      T     "MAL1S032Par".Par.ParIntProcess.Speed_ILO_Fan;
F04a: NOP   0;

IO4:  NOP   0;
      NOP   0;
// --- FCM 05 - Fans with target air temperature ---
      L     "MAL1S032Par".Ilo.ILOMode;
      L     5;
      <>I   ;
      SPB   IO5;
// man on
      U     "MAL1S032Par".Ilo.GrCMDManOn[1];
      S     "G271M".Gr.InManual; // FAN KILN 1
      S     "G273M".Gr.InManual; // RECYCLING AIR LOUVER KILN 1
      S     "G273M".Gr.CmdOn; // No Button: RECYCLING AIR LOUVER KILN 1
      S     "G273M".Gr.CmdContinue; // No Button RECYCLING AIR LOUVER KILN 1
      S     "G276M".Gr.InManual; // HEATING KILN 1
      S     "G276M".Gr.CmdOn; // No Button: HEATING KILN 1
      S     "G276M".Gr.CmdContinue; // No Button HEATING KILN 1
      S     "G277M".Gr.InManual; // LOUVER AIR HEATER 1 FOR KILN 1
      S     "G277M".Gr.CmdOn; // No Button: LOUVER AIR HEATER 1 FOR KILN 1
      S     "G277M".Gr.CmdContinue; // No Button LOUVER AIR HEATER 1 FOR KILN 1
      S     "G272M".Gr.InManual; // FRESH AIR LOUVER KILN 1
      S     "G272M".Gr.CmdOn; // No Button: FRESH AIR LOUVER KILN 1
      S     "G272M".Gr.CmdContinue; // No Button FRESH AIR LOUVER KILN 1
      S     "G278M".Gr.InManual; // WITHERING AIR KILN 1
      S     "G278M".Gr.CmdOn; // No Button: WITHERING AIR KILN 1
      S     "G278M".Gr.CmdContinue; // No Button WITHERING AIR KILN 1
      R     "MAL1S032Par".Ilo.GrCMDManOn[1];
// man off
      U     "MAL1S032Par".Ilo.GrCMDManOff[1];
      S     "G271M".Gr.CmdManualOff; // FAN KILN 1
      R     "G271M".Gr.InManual; // FAN KILN 1
      R     "G271M".USW14; // ILO-cmd
      R     "G271M".USW15; // ILO-cmd
      S     "G273M".Gr.CmdManualOff; // RECYCLING AIR LOUVER KILN 1
      R     "G273M".Gr.InManual; // RECYCLING AIR LOUVER KILN 1
      R     "G273M".USW14; // ILO-cmd
      R     "G273M".USW15; // ILO-cmd
      S     "G276M".Gr.CmdManualOff; // HEATING KILN 1
      R     "G276M".Gr.InManual; // HEATING KILN 1
      R     "G276M".USW14; // ILO-cmd
      R     "G276M".USW15; // ILO-cmd
      S     "G277M".Gr.CmdManualOff; // LOUVER AIR HEATER 1 FOR KILN 1
      R     "G277M".Gr.InManual; // LOUVER AIR HEATER 1 FOR KILN 1
      R     "G277M".USW14; // ILO-cmd
      R     "G277M".USW15; // ILO-cmd
      S     "G272M".Gr.CmdManualOff; // FRESH AIR LOUVER KILN 1
      R     "G272M".Gr.InManual; // FRESH AIR LOUVER KILN 1
      R     "G272M".USW14; // ILO-cmd
      R     "G272M".USW15; // ILO-cmd
      S     "G278M".Gr.CmdManualOff; // WITHERING AIR KILN 1
      R     "G278M".Gr.InManual; // WITHERING AIR KILN 1
      R     "G278M".USW14; // ILO-cmd
      R     "G278M".USW15; // ILO-cmd
      R     "MAL1S032Par".Ilo.GrCMDManOff[1];
      R     "MAL1S032Par".Ilo.GrCMDManAdditional.Cmd1[1];
      R     "MAL1S032Par".Ilo.GrCMDManAdditional.Cmd2[1];
// man start
      U     "MAL1S032Par".Ilo.GrCMDManStart[1];
      S     "G271M".Gr.CmdOn; // FAN KILN 1
      S     "G271M".Gr.CmdContinue; // FAN KILN 1
      S     "G273M".Gr.CmdOn; // RECYCLING AIR LOUVER KILN 1
      S     "G273M".Gr.CmdContinue; // RECYCLING AIR LOUVER KILN 1
      S     "G276M".Gr.CmdOn; // HEATING KILN 1
      S     "G276M".Gr.CmdContinue; // HEATING KILN 1
      S     "G277M".Gr.CmdOn; // LOUVER AIR HEATER 1 FOR KILN 1
      S     "G277M".Gr.CmdContinue; // LOUVER AIR HEATER 1 FOR KILN 1
      S     "G272M".Gr.CmdOn; // FRESH AIR LOUVER KILN 1
      S     "G272M".Gr.CmdContinue; // FRESH AIR LOUVER KILN 1
      S     "G278M".Gr.CmdOn; // WITHERING AIR KILN 1
      S     "G278M".Gr.CmdContinue; // WITHERING AIR KILN 1
      R     "MAL1S032Par".Ilo.GrCMDManStart[1];
      U     "MAL1S032Par".Ilo.GrCMDManStart[2];
      R     "MAL1S032Par".Ilo.GrCMDManStart[2];
// man stop
      U     "MAL1S032Par".Ilo.GrSTMan[17];
      S     "G271M".Gr.CmdOff; // FAN KILN 1
      S     "G273M".Gr.CmdOff; // RECYCLING AIR LOUVER KILN 1
      S     "G276M".Gr.CmdOff; // HEATING KILN 1
      S     "G277M".Gr.CmdOff; // LOUVER AIR HEATER 1 FOR KILN 1
      S     "G272M".Gr.CmdOff; // FRESH AIR LOUVER KILN 1
      S     "G278M".Gr.CmdOff; // WITHERING AIR KILN 1
      R     "MAL1S032Par".Ilo.GrSTMan[17];
// man fault reset
      U     "MAL1S032Par".Ilo.GrCMDManFaultReset[1];
      S     "G271M".Gr.CmdFaultReset; // FAN KILN 1
      S     "G273M".Gr.CmdFaultReset; // RECYCLING AIR LOUVER KILN 1
      S     "G276M".Gr.CmdFaultReset; // HEATING KILN 1
      S     "G277M".Gr.CmdFaultReset; // LOUVER AIR HEATER 1 FOR KILN 1
      S     "G272M".Gr.CmdFaultReset; // FRESH AIR LOUVER KILN 1
      S     "G278M".Gr.CmdFaultReset; // WITHERING AIR KILN 1
      R     "MAL1S032Par".Ilo.GrCMDManFaultReset[1];
// target position
      UN    "G271M".Gr.InManual; // FAN KILN 1
      O(    ;
      L     "MAL1S032Par".Ilo.Code_ILO_Funktion0;
      L     500;
      <>I   ;
      )     ;
      SPB   F05b;
      L     "MAL1S032Par".Ilo.SetpointInt01[1];
      T     "MAL1S032Par".Par.ParIntProcess.Speed_ILO_Fan;
F05b: NOP   0;
      UN    "G273M".Gr.InManual; // Recycling Air Flap Kilningbox 1
      O(    ;
      L     "MAL1S032Par".Ilo.Code_ILO_Funktion0;
      L     500;
      <>I   ;
      )     ;
      SPB   F05c;
      L     "MAL1S032Par".Ilo.SetpointInt03[1];
      T     "MAL1S032Par".Par.ParIntProcess.TarPos_ILO_RecycAir;
F05c: NOP   0;
      UN    "G278M".Gr.InManual; // Withering Air Flap Kilningbox 1
      O(    ;
      L     "MAL1S032Par".Ilo.Code_ILO_Funktion0;
      L     500;
      <>I   ;
      )     ;
      SPB   F05d;
      L     "MAL1S032Par".Ilo.SetpointInt04[1];
      T     "MAL1S032Par".Par.ParIntProcess.TarPos_ILO_WitheringAir;
F05d: NOP   0;
      UN    "G276M".Gr.InManual; // Heating Kiln 1
      O(    ;
      L     "MAL1S032Par".Ilo.Code_ILO_Funktion0;
      L     500;
      <>I   ;
      )     ;
      SPB   F05e;
      L     "MAL1S032Par".Ilo.SetpointInt01[2];
      T     "MAL1S032Par".Par.ParIntProcess.TargetTemperature_ILO;
F05e: NOP   0;

IO5:  NOP   0;
      NOP   0;
// --- FCM 06 - Fresh air flap ---
      L     "MAL1S032Par".Ilo.ILOMode;
      L     6;
      <>I   ;
      SPB   IO6;
// man on
      U     "MAL1S032Par".Ilo.GrCMDManOn[1];
      S     "G272M".Gr.InManual; // FRESH AIR LOUVER KILN 1
      R     "MAL1S032Par".Ilo.GrCMDManOn[1];
// man off
      U     "MAL1S032Par".Ilo.GrCMDManOff[1];
      S     "G272M".Gr.CmdManualOff; // FRESH AIR LOUVER KILN 1
      R     "G272M".Gr.InManual; // FRESH AIR LOUVER KILN 1
      R     "G272M".USW14; // ILO-cmd
      R     "G272M".USW15; // ILO-cmd
      R     "MAL1S032Par".Ilo.GrCMDManOff[1];
      R     "MAL1S032Par".Ilo.GrCMDManAdditional.Cmd1[1];
      R     "MAL1S032Par".Ilo.GrCMDManAdditional.Cmd2[1];
// man start
      U     "MAL1S032Par".Ilo.GrCMDManStart[1];
      S     "G272M".Gr.CmdOn; // FRESH AIR LOUVER KILN 1
      S     "G272M".Gr.CmdContinue; // FRESH AIR LOUVER KILN 1
      R     "MAL1S032Par".Ilo.GrCMDManStart[1];
      U     "MAL1S032Par".Ilo.GrCMDManStart[2];
      R     "MAL1S032Par".Ilo.GrCMDManStart[2];
// man stop
      U     "MAL1S032Par".Ilo.GrCMDManStop[1];
      S     "G272M".Gr.CmdOff; // FRESH AIR LOUVER KILN 1
      R     "MAL1S032Par".Ilo.GrCMDManStop[1];
// man fault reset
      U     "MAL1S032Par".Ilo.GrCMDManFaultReset[1];
      S     "G272M".Gr.CmdFaultReset; // FRESH AIR LOUVER KILN 1
      R     "MAL1S032Par".Ilo.GrCMDManFaultReset[1];
// moving direction

// target position
      UN    "G272M".Gr.InManual; // FRESH AIR LOUVER KILN 1
      SPB   F06b;
      L     "MAL1S032Par".Ilo.SetpointInt01[1];
      T     "MAL1S032Par".Par.ParIntProcess.TarPos_ILO_FreshAir;
F06b: NOP   0;

IO6:  NOP   0;
      NOP   0;
// --- FCM 07 - Recycling air flap ---
      L     "MAL1S032Par".Ilo.ILOMode;
      L     7;
      <>I   ;
      SPB   IO7;
// man on
      U     "MAL1S032Par".Ilo.GrCMDManOn[1];
      S     "G273M".Gr.InManual; // RECYCLING AIR LOUVER KILN 1
      S     "G278M".Gr.InManual; // WITHERING AIR KILN 1
      R     "MAL1S032Par".Ilo.GrCMDManOn[1];
// man off
      U     "MAL1S032Par".Ilo.GrCMDManOff[1];
      S     "G273M".Gr.CmdManualOff; // RECYCLING AIR LOUVER KILN 1
      R     "G273M".Gr.InManual; // RECYCLING AIR LOUVER KILN 1
      R     "G273M".USW14; // ILO-cmd
      R     "G273M".USW15; // ILO-cmd
      S     "G278M".Gr.CmdManualOff; // WITHERING AIR KILN 1
      R     "G278M".Gr.InManual; // WITHERING AIR KILN 1
      R     "G278M".USW14; // ILO-cmd
      R     "G278M".USW15; // ILO-cmd
      R     "MAL1S032Par".Ilo.GrCMDManOff[1];
      R     "MAL1S032Par".Ilo.GrCMDManAdditional.Cmd1[1];
      R     "MAL1S032Par".Ilo.GrCMDManAdditional.Cmd2[1];
// man start
      U     "MAL1S032Par".Ilo.GrCMDManStart[1];
      S     "G273M".Gr.CmdOn; // RECYCLING AIR LOUVER KILN 1
      S     "G273M".Gr.CmdContinue; // RECYCLING AIR LOUVER KILN 1
      S     "G278M".Gr.CmdOn; // WITHERING AIR KILN 1
      S     "G278M".Gr.CmdContinue; // WITHERING AIR KILN 1
      R     "MAL1S032Par".Ilo.GrCMDManStart[1];
      U     "MAL1S032Par".Ilo.GrCMDManStart[2];
      R     "MAL1S032Par".Ilo.GrCMDManStart[2];
// man stop
      U     "MAL1S032Par".Ilo.GrCMDManStop[1];
      S     "G273M".Gr.CmdOff; // RECYCLING AIR LOUVER KILN 1
      S     "G278M".Gr.CmdOff; // WITHERING AIR KILN 1
      R     "MAL1S032Par".Ilo.GrCMDManStop[1];
// man fault reset
      U     "MAL1S032Par".Ilo.GrCMDManFaultReset[1];
      S     "G273M".Gr.CmdFaultReset; // RECYCLING AIR LOUVER KILN 1
      S     "G278M".Gr.CmdFaultReset; // WITHERING AIR KILN 1
      R     "MAL1S032Par".Ilo.GrCMDManFaultReset[1];
// moving direction

// target position
      UN    "G273M".Gr.InManual; // RECYCLING AIR LOUVER KILN 1
      SPB   F07a;
      L     "MAL1S032Par".Ilo.SetpointInt01[1];
      T     "MAL1S032Par".Par.ParIntProcess.TarPos_ILO_RecycAir;
F07a: NOP   0;
IO7:  NOP   0;
      NOP   0;
// --- FCM 09 - Floor drives ---
      L     "MAL1S032Par".Ilo.ILOMode;
      L     9;
      <>I   ;
      SPB   IO9;
// man on
      U     "MAL1S032Par".Ilo.GrCMDManOn[1];
      S     "G266M".Gr.InManual; // TRAVELLING DRIVE KILN 1
      R     "MAL1S032Par".Ilo.GrCMDManOn[1];
// man off
      U     "MAL1S032Par".Ilo.GrCMDManOff[1];
      S     "G266M".Gr.CmdManualOff; // TRAVELLING DRIVE KILN 1
      R     "G266M".Gr.InManual; // TRAVELLING DRIVE KILN 1
      R     "G266M".USW14; // ILO-cmd
      R     "G266M".USW15; // ILO-cmd
      R     "MAL1S032Par".Ilo.GrCMDManOff[1];
      R     "MAL1S032Par".Ilo.GrCMDManAdditional.Cmd1[1];
      R     "MAL1S032Par".Ilo.GrCMDManAdditional.Cmd2[1];
// man start
      U     "MAL1S032Par".Ilo.GrCMDManStart[1];
      S     "G266M".Gr.CmdOn; // TRAVELLING DRIVE KILN 1
      S     "G266M".Gr.CmdContinue; // TRAVELLING DRIVE KILN 1
      R     "MAL1S032Par".Ilo.GrCMDManStart[1];
      U     "MAL1S032Par".Ilo.GrCMDManStart[2];
      R     "MAL1S032Par".Ilo.GrCMDManStart[2];
// man stop
      U     "MAL1S032Par".Ilo.GrCMDManStop[1];
      S     "G266M".Gr.CmdOff; // TRAVELLING DRIVE KILN 1
      R     "MAL1S032Par".Ilo.GrCMDManStop[1];
// man fault reset
      U     "MAL1S032Par".Ilo.GrCMDManFaultReset[1];
      S     "G266M".Gr.CmdFaultReset; // TRAVELLING DRIVE KILN 1
      R     "MAL1S032Par".Ilo.GrCMDManFaultReset[1];
      NOP   0;
      UN    "G266M".Gr.InManual; // TRAVELLING DRIVE KILN 1
      O     ;
      UN    "MAL1S032Par".Ilo.GrCMDManAdditional.Cmd1[1];
      UN    "MAL1S032Par".Ilo.GrCMDManAdditional.Cmd2[1];
      SPB   f092;
      U     "MAL1S032Par".Ilo.GrCMDManAdditional.Cmd1[1];
      =     "G266M".USW14; // ILO-cmd run fwd
      U     "MAL1S032Par".Ilo.GrCMDManAdditional.Cmd2[1];
      =     "G266M".USW15; // ILO-cmd run rev
// target position
      L     "MAL1S032Par".Ilo.SetpointInt01[1];
      T     "MAL1S032Par".Par.ParIntProcess.Speed_ILO_FloorRotating;
f092: NOP   0;

IO9:  NOP   0;
      NOP   0;
// --- FCM 10 - Floor drives and lifting devices ---
      L     "MAL1S032Par".Ilo.ILOMode;
      L     10;
      <>I   ;
      SPB   IO10;
// man on
      U     "MAL1S032Par".Ilo.GrCMDManOn[1];
      S     "G265M".Gr.InManual; // LIFTING DEVICE KILN 1
      S     "G265M".Gr.CmdOn; // No Button: LIFTING DEVICE KILN 1
      S     "G265M".Gr.CmdContinue; // No Button LIFTING DEVICE KILN 1
      S     "G266M".Gr.InManual; // TRAVELLING DRIVE KILN 1
      R     "MAL1S032Par".Ilo.GrCMDManOn[1];
// man off
      U     "MAL1S032Par".Ilo.GrCMDManOff[1];
      S     "G265M".Gr.CmdManualOff; // LIFTING DEVICE KILN 1
      R     "G265M".Gr.InManual; // LIFTING DEVICE KILN 1
      R     "G265M".USW14; // ILO-cmd
      R     "G265M".USW15; // ILO-cmd
      S     "G266M".Gr.CmdManualOff; // TRAVELLING DRIVE KILN 1
      R     "G266M".Gr.InManual; // TRAVELLING DRIVE KILN 1
      R     "G266M".USW14; // ILO-cmd
      R     "G266M".USW15; // ILO-cmd
      R     "MAL1S032Par".Ilo.GrCMDManOff[1];
      R     "MAL1S032Par".Ilo.GrCMDManAdditional.Cmd1[1];
      R     "MAL1S032Par".Ilo.GrCMDManAdditional.Cmd2[1];
// man start
      U     "MAL1S032Par".Ilo.GrCMDManStart[1];
      S     "G266M".Gr.CmdOn; // TRAVELLING DRIVE KILN 1
      S     "G266M".Gr.CmdContinue; // TRAVELLING DRIVE KILN 1
      R     "MAL1S032Par".Ilo.GrCMDManStart[1];
      U     "MAL1S032Par".Ilo.GrCMDManStart[2];
      S     "G265M".Gr.CmdOn; // LIFTING DEVICE KILN 1
      S     "G265M".Gr.CmdContinue; // LIFTING DEVICE KILN 1
      R     "MAL1S032Par".Ilo.GrCMDManStart[2];
      U     "MAL1S032Par".Ilo.GrCMDManStart[3];
      R     "MAL1S032Par".Ilo.GrCMDManStart[3];
// man stop
      U     "MAL1S032Par".Ilo.GrCMDManStop[1];
      S     "G265M".Gr.CmdOff; // LIFTING DEVICE KILN 1
      S     "G266M".Gr.CmdOff; // TRAVELLING DRIVE KILN 1
      R     "MAL1S032Par".Ilo.GrCMDManStop[1];
// man fault reset
      U     "MAL1S032Par".Ilo.GrCMDManFaultReset[1];
      S     "G265M".Gr.CmdFaultReset; // LIFTING DEVICE KILN 1
      S     "G266M".Gr.CmdFaultReset; // TRAVELLING DRIVE KILN 1
      R     "MAL1S032Par".Ilo.GrCMDManFaultReset[1];
// moving direction
      NOP   0;
      UN    "G266M".Gr.InManual; // TRAVELLING DRIVE KILN 1
      O     ;
      UN    "MAL1S032Par".Ilo.GrCMDManAdditional.Cmd1[1];
      UN    "MAL1S032Par".Ilo.GrCMDManAdditional.Cmd2[1];
      SPB   f102;
      U     "MAL1S032Par".Ilo.GrCMDManAdditional.Cmd1[1];
      =     "G266M".USW14; // ILO-cmd run fwd
      U     "MAL1S032Par".Ilo.GrCMDManAdditional.Cmd2[1];
      =     "G266M".USW15; // ILO-cmd run rev
// target speed floor drives
      L     "MAL1S032Par".Ilo.SetpointInt01[1];
      T     "MAL1S032Par".Par.ParIntProcess.Speed_ILO_FloorRotating;
f102: NOP   0;
      UN    "G265M".Gr.InManual; // LIFTING DEVICE KILN 1
      O(    ;
      L     "MAL1S032Par".Ilo.Code_ILO_Funktion0;
      L     1000;
      <>I   ;
      )     ;
      SPB   f103;
// target position lifting devices
      L     "MAL1S032Par".Ilo.SetpointInt02[1];
      T     "MAL1S032Par".Par.ParIntProcess.TarPos_ILO_LiftDev;
f103: NOP   0;

IO10: NOP   0;
      NOP   0;
// --- FCM 11 - Floor drives and lifting devices and screw ---
      L     "MAL1S032Par".Ilo.ILOMode;
      L     11;
      <>I   ;
      SPB   IO11;
// man on
      U     "MAL1S032Par".Ilo.GrCMDManOn[1];
      S     "G265M".Gr.InManual; // LIFTING DEVICE KILN 1
      S     "G265M".Gr.CmdOn; // No Button: LIFTING DEVICE KILN 1
      S     "G265M".Gr.CmdContinue; // No Button LIFTING DEVICE KILN 1
      S     "G266M".Gr.InManual; // TRAVELLING DRIVE KILN 1
      S     "G267M".Gr.InManual; // UNLOADING / LOADING SCREW KILN 1
      R     "MAL1S032Par".Ilo.GrCMDManOn[1];
// man off
      U     "MAL1S032Par".Ilo.GrCMDManOff[1];
      S     "G265M".Gr.CmdManualOff; // LIFTING DEVICE KILN 1
      R     "G265M".Gr.InManual; // LIFTING DEVICE KILN 1
      R     "G265M".USW14; // ILO-cmd
      R     "G265M".USW15; // ILO-cmd
      S     "G266M".Gr.CmdManualOff; // TRAVELLING DRIVE KILN 1
      R     "G266M".Gr.InManual; // TRAVELLING DRIVE KILN 1
      R     "G266M".USW14; // ILO-cmd
      R     "G266M".USW15; // ILO-cmd
      S     "G267M".Gr.CmdManualOff; // UNLOADING / LOADING SCREW KILN 1
      R     "G267M".Gr.InManual; // UNLOADING / LOADING SCREW KILN 1
      R     "G267M".USW14; // ILO-cmd
      R     "G267M".USW15; // ILO-cmd
      R     "MAL1S032Par".Ilo.GrCMDManOff[1];
      R     "MAL1S032Par".Ilo.GrCMDManAdditional.Cmd1[1];
      R     "MAL1S032Par".Ilo.GrCMDManAdditional.Cmd2[1];
// man start
      U     "MAL1S032Par".Ilo.GrCMDManStart[1];
      S     "G266M".Gr.CmdOn; // TRAVELLING DRIVE KILN 1
      S     "G266M".Gr.CmdContinue; // TRAVELLING DRIVE KILN 1
      R     "MAL1S032Par".Ilo.GrCMDManStart[1];
      U     "MAL1S032Par".Ilo.GrCMDManStart[2];
      S     "G265M".Gr.CmdOn; // LIFTING DEVICE KILN 1
      S     "G265M".Gr.CmdContinue; // LIFTING DEVICE KILN 1
      R     "MAL1S032Par".Ilo.GrCMDManStart[2];
      U     "MAL1S032Par".Ilo.GrCMDManStart[3];
      S     "G267M".Gr.CmdOn; // UNLOADING / LOADING SCREW KILN 1
      S     "G267M".Gr.CmdContinue; // UNLOADING / LOADING SCREW KILN 1
      R     "MAL1S032Par".Ilo.GrCMDManStart[3];
      U     "MAL1S032Par".Ilo.GrCMDManStart[4];
      S     "G267M".Gr.CmdOn; // UNLOADING / LOADING SCREW KILN 1
      S     "G267M".Gr.CmdContinue; // UNLOADING / LOADING SCREW KILN 1
      R     "MAL1S032Par".Ilo.GrCMDManStart[4];
// man stop
      U     "MAL1S032Par".Ilo.GrCMDManStop[1];
      S     "G265M".Gr.CmdOff; // LIFTING DEVICE KILN 1
      S     "G266M".Gr.CmdOff; // TRAVELLING DRIVE KILN 1
      S     "G267M".Gr.CmdOff; // UNLOADING / LOADING SCREW KILN 1
      R     "MAL1S032Par".Ilo.GrCMDManStop[1];
// man fault reset
      U     "MAL1S032Par".Ilo.GrCMDManFaultReset[1];
      S     "G265M".Gr.CmdFaultReset; // LIFTING DEVICE KILN 1
      S     "G266M".Gr.CmdFaultReset; // TRAVELLING DRIVE KILN 1
      S     "G267M".Gr.CmdFaultReset; // UNLOADING / LOADING SCREW KILN 1
      R     "MAL1S032Par".Ilo.GrCMDManFaultReset[1];
// moving direction
      UN    "G266M".Gr.InManual; // TRAVELLING DRIVE KILN 1
      O     ;
      UN    "MAL1S032Par".Ilo.GrCMDManAdditional.Cmd1[1];
      UN    "MAL1S032Par".Ilo.GrCMDManAdditional.Cmd2[1];
      SPB   f112;
      U     "MAL1S032Par".Ilo.GrCMDManAdditional.Cmd1[1];
      =     "G266M".USW14; // ILO-cmd run fwd
      U     "MAL1S032Par".Ilo.GrCMDManAdditional.Cmd2[1];
      =     "G266M".USW15; // ILO-cmd run rev
// target speed floor drives
      L     "MAL1S032Par".Ilo.SetpointInt01[1];
      T     "MAL1S032Par".Par.ParIntProcess.Speed_ILO_FloorRotating;
f112: NOP   0;
      UN    "G265M".Gr.InManual; // Malting Plant OAO Belsolod Ivanonvo Weissrussland
      O(    ;
      L     "MAL1S032Par".Ilo.Code_ILO_Funktion0;
      L     1100;
      <>I   ;
      )     ;
      SPB   f113;
// target position lifting devices
      L     "MAL1S032Par".Ilo.SetpointInt01[2];
      L     "MAL1S032Par".Ilo.SetpointInt02[1];
      T     "MAL1S032Par".Par.ParIntProcess.TarPos_ILO_LiftDev;
f113: NOP   0;
      UN    "G267M".Gr.InManual; // UNLOADING / LOADING SCREW KILN 1
      O     ;
      UN    "MAL1S032Par".Ilo.GrCMDManAdditional.Cmd1[3];
      UN    "MAL1S032Par".Ilo.GrCMDManAdditional.Cmd2[3];
      SPB   f114;
      U     "MAL1S032Par".Ilo.GrCMDManAdditional.Cmd1[3];
      =     "G267M".USW14; // ILO-cmd run fwd
      U     "MAL1S032Par".Ilo.GrCMDManAdditional.Cmd2[3];
      =     "G267M".USW15; // ILO-cmd run rev
f114: NOP   0;
IO11: NOP   0;
      NOP   0;
// --- FCM 12 - Floor drives and lifting devices and screw and discharging flap ---
      L     "MAL1S032Par".Ilo.ILOMode;
      L     12;
      <>I   ;
      SPB   IO12;
// man on
      U     "MAL1S032Par".Ilo.GrCMDManOn[1];
      S     "G265M".Gr.InManual; // LIFTING DEVICE KILN 1
      S     "G265M".Gr.CmdOn; // No Button: LIFTING DEVICE KILN 1
      S     "G265M".Gr.CmdContinue; // No Button LIFTING DEVICE KILN 1
      S     "G266M".Gr.InManual; // TRAVELLING DRIVE KILN 1
      S     "G267M".Gr.InManual; // UNLOADING / LOADING SCREW KILN 1
      S     "G268M".Gr.InManual; // DISCHARGE DOOR KILN 1
      R     "MAL1S032Par".Ilo.GrCMDManOn[1];
// man off
      U     "MAL1S032Par".Ilo.GrCMDManOff[1];
      S     "G265M".Gr.CmdManualOff; // LIFTING DEVICE KILN 1
      R     "G265M".Gr.InManual; // LIFTING DEVICE KILN 1
      R     "G265M".USW14; // ILO-cmd
      R     "G265M".USW15; // ILO-cmd
      S     "G266M".Gr.CmdManualOff; // TRAVELLING DRIVE KILN 1
      R     "G266M".Gr.InManual; // TRAVELLING DRIVE KILN 1
      R     "G266M".USW14; // ILO-cmd
      R     "G266M".USW15; // ILO-cmd
      S     "G267M".Gr.CmdManualOff; // UNLOADING / LOADING SCREW KILN 1
      R     "G267M".Gr.InManual; // UNLOADING / LOADING SCREW KILN 1
      R     "G267M".USW14; // ILO-cmd
      R     "G267M".USW15; // ILO-cmd
      S     "G268M".Gr.CmdManualOff; // DISCHARGE DOOR KILN 1
      R     "G268M".Gr.InManual; // DISCHARGE DOOR KILN 1
      R     "G268M".USW14; // ILO-cmd
      R     "G268M".USW15; // ILO-cmd
      R     "MAL1S032Par".Ilo.GrCMDManOff[1];
      R     "MAL1S032Par".Ilo.GrCMDManAdditional.Cmd1[1];
      R     "MAL1S032Par".Ilo.GrCMDManAdditional.Cmd2[1];
// man start
      U     "MAL1S032Par".Ilo.GrCMDManStart[1];
      S     "G266M".Gr.CmdOn; // TRAVELLING DRIVE KILN 1
      S     "G266M".Gr.CmdContinue; // TRAVELLING DRIVE KILN 1
      R     "MAL1S032Par".Ilo.GrCMDManStart[1];
      U     "MAL1S032Par".Ilo.GrCMDManStart[2];
      S     "G265M".Gr.CmdOn; // LIFTING DEVICE KILN 1
      S     "G265M".Gr.CmdContinue; // LIFTING DEVICE KILN 1
      R     "MAL1S032Par".Ilo.GrCMDManStart[2];
      U     "MAL1S032Par".Ilo.GrCMDManStart[3];
      S     "G267M".Gr.CmdOn; // UNLOADING / LOADING SCREW KILN 1
      S     "G267M".Gr.CmdContinue; // UNLOADING / LOADING SCREW KILN 1
      R     "MAL1S032Par".Ilo.GrCMDManStart[3];
      U     "MAL1S032Par".Ilo.GrCMDManStart[4];
      S     "G267M".Gr.CmdOn; // UNLOADING / LOADING SCREW KILN 1
      S     "G267M".Gr.CmdContinue; // UNLOADING / LOADING SCREW KILN 1
      R     "MAL1S032Par".Ilo.GrCMDManStart[4];
// man stop
      U     "MAL1S032Par".Ilo.GrCMDManStop[1];
      S     "G265M".Gr.CmdOff; // LIFTING DEVICE KILN 1
      S     "G266M".Gr.CmdOff; // TRAVELLING DRIVE KILN 1
      S     "G267M".Gr.CmdOff; // UNLOADING / LOADING SCREW KILN 1
      S     "G268M".Gr.CmdOff; // DISCHARGE DOOR KILN 1
      R     "MAL1S032Par".Ilo.GrCMDManStop[1];
// man fault reset
      U     "MAL1S032Par".Ilo.GrCMDManFaultReset[1];
      S     "G265M".Gr.CmdFaultReset; // LIFTING DEVICE KILN 1
      S     "G266M".Gr.CmdFaultReset; // TRAVELLING DRIVE KILN 1
      S     "G267M".Gr.CmdFaultReset; // UNLOADING / LOADING SCREW KILN 1
      S     "G268M".Gr.CmdFaultReset; // DISCHARGE DOOR KILN 1
      R     "MAL1S032Par".Ilo.GrCMDManFaultReset[1];
// moving direction
      UN    "G266M".Gr.InManual; // TRAVELLING DRIVE KILN 1
      O     ;
      UN    "MAL1S032Par".Ilo.GrCMDManAdditional.Cmd1[1];
      UN    "MAL1S032Par".Ilo.GrCMDManAdditional.Cmd2[1];
      SPB   f122;
      U     "MAL1S032Par".Ilo.GrCMDManAdditional.Cmd1[1];
      =     "G266M".USW14; // ILO-cmd run fwd
      U     "MAL1S032Par".Ilo.GrCMDManAdditional.Cmd2[1];
      =     "G266M".USW15; // ILO-cmd run rev
// target speed floor drives
      L     "MAL1S032Par".Ilo.SetpointInt01[1];
      T     "MAL1S032Par".Par.ParIntProcess.Speed_ILO_FloorRotating;
f122: NOP   0;
      UN    "G265M".Gr.InManual; // LIFTING DEVICE KILN 1
      O(    ;
      L     "MAL1S032Par".Ilo.Code_ILO_Funktion0;
      L     1200;
      <>I   ;
      )     ;
      SPB   f123;
// target position lifting devices
      L     "MAL1S032Par".Ilo.SetpointInt02[1];
      T     "MAL1S032Par".Par.ParIntProcess.TarPos_ILO_LiftDev;
f123: NOP   0;
      UN    "G267M".Gr.InManual; // Malting Plant OAO Belsolod Ivanonvo Weissrussland
      O     ;
      UN    "MAL1S032Par".Ilo.GrCMDManAdditional.Cmd1[3];
      UN    "MAL1S032Par".Ilo.GrCMDManAdditional.Cmd2[3];
      SPB   f124;
      U     "MAL1S032Par".Ilo.GrCMDManAdditional.Cmd1[3];
      =     "G267M".USW14; // ILO-cmd run fwd
      U     "MAL1S032Par".Ilo.GrCMDManAdditional.Cmd2[3];
      =     "G267M".USW15; // ILO-cmd run rev
f124: NOP   0;
      UN    "G268M".Gr.InManual; // DISCHARGE DOOR KILN 1
      O     ;
      UN    "MAL1S032Par".Ilo.GrCMDManAdditional.Cmd1[4];
      UN    "MAL1S032Par".Ilo.GrCMDManAdditional.Cmd2[4];
      SPB   f125;
      U     "MAL1S032Par".Ilo.GrCMDManAdditional.Cmd1[4];
      =     "G268M".USW14; // ILO-cmd OPEN
      U     "MAL1S032Par".Ilo.GrCMDManAdditional.Cmd2[4];
      =     "G268M".USW15; // ILO-cmd CLOSE
f125: NOP   0;
IO12: NOP   0;
//
// copy state
      U     "G265M".Gr.InOutAutostartMan; // LIFTING DEVICE KILN 1
      =     "MAL1S032Par".Ilo.GrSTMan[1];
      U     "G266M".Gr.InOutAutostartMan; // TRAVELLING DRIVE KILN 1
      =     "MAL1S032Par".Ilo.GrSTMan[2];
      U     "G267M".Gr.InOutAutostartMan; // UNLOADING / LOADING SCREW KILN 1
      =     "MAL1S032Par".Ilo.GrSTMan[3];
      U     "G268M".Gr.InOutAutostartMan; // DISCHARGE DOOR KILN 1
      =     "MAL1S032Par".Ilo.GrSTMan[4];
      U     "G271M".Gr.InOutAutostartMan; // FAN KILN 1
      =     "MAL1S032Par".Ilo.GrSTMan[6];
      U     "G276M".Gr.InOutAutostartMan; // HEATING KILN 1
      =     "MAL1S032Par".Ilo.GrSTMan[11];
      U     "G277M".Gr.InOutAutostartMan; // LOUVER AIR HEATER 1 FOR KILN 1
      =     "MAL1S032Par".Ilo.GrSTMan[12];
      U     "G272M".Gr.InOutAutostartMan; // FRESH AIR LOUVER KILN 1
      =     "MAL1S032Par".Ilo.GrSTMan[13];
      U     "G278M".Gr.InOutAutostartMan; // WITHERING AIR KILN 1
      =     "MAL1S032Par".Ilo.GrSTMan[14];
      U     "G273M".Gr.InOutAutostartMan; // RECYCLING AIR LOUVER KILN 1
      =     "MAL1S032Par".Ilo.GrSTMan[15];
      U     "G279M".Gr.InOutAutostartMan; // HEATING KILN 1 + 2
      =     "MAL1S032Par".Ilo.GrSTMan[16];
NETWORK
TITLE =ASW_9999: Init Flag
// clear all flags explicde to find them back
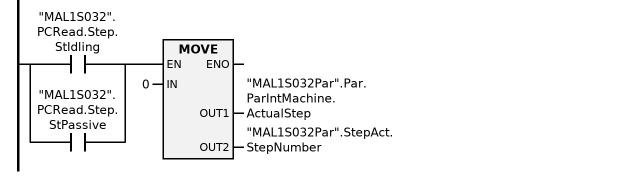
      U     "MAL1S032".PCRead.Step.StIdling;
      O     "MAL1S032".PCRead.Step.StPassive;
      R     "MAL1S032Par".Par.FlagFunction_1.StepLoading;
      R     "MAL1S032Par".Par.FlagFunction_1.StepUnloading;
      R     "MAL1S032Par".Par.FlagFunction_1.StepCleaning;
      R     "MAL1S032Par".Par.FlagFunction_1.LoadingBreak;
      R     "MAL1S032Par".Par.FlagFunction_1.UnloadingBreak;
      R     "MAL1S032Par".Par.FlagFunction_1.CleaningBreak;
      R     "MAL1S032Par".Par.FlagFunction_1.FinishLoading;
      R     "MAL1S032Par".Par.FlagFunction_1.FinishUnloading;
      R     "MAL1S032Par".Par.FlagFunction_1.FinishCleaning;
      R     "MAL1S032Par".Par.FlagFunction_1.Entladerunden_erreicht;
      R     "MAL1S032Par".Par.FlagFunction_1.Reinigungsrunde_erreicht;
      R     "MAL1S032Par".Par.FlagFunction_1.UnloadEnd;
      R     "MAL1S032Par".Par.FlagFunction_1.LoadEnd;
      R     "MAL1S032Par".Par.FlagFunction_1.UnloadFirstPart;
      R     "MAL1S032Par".Par.FlagFunction_1.UnloadSecondPart;
      R     "MAL1S032Par".Par.FlagProcess.ProcessActive;
      R     "MAL1S032Par".Par.FlagProcess.StartProzess_FP;
      R     "MAL1S032Par".Par.FlagProcess.StartProzess_SCAN;
      R     "MAL1S032Par".Par.FlagProcess.TurningFloor;
      R     "MAL1S032Par".Par.FlagProcess.Cooling_Activ;
      R     "MAL1S032Par".Par.FlagProcess.FP_SendResultToPIC;
      R     "MAL1S032Par".Par.FlagProcess.ProcessEnd;

// --> Wie bei Bank Avangard
      U     "MAL1S032".PCRead.Step.StPassive;
      R     "MAL1S032Par".Par.FlagMachine.WEGMESSUNG_0_FLAG;
      R     "MAL1S032Par".Par.FlagMachine.ImpulsNullstellung;
      R     "MAL1S032Par".Par.FlagMachine.CmdTurnFwdAfterLoading;
      R     "MAL1S032Par".Par.FlagMachine.CmdTurnRevAfterLoading;
      R     "MAL1S032Par".Par.FlagMachine.ImpulsNullstellungFP;
      R     "MAL1S032Par".Par.FlagMachine.CmdTurnFwdAfterTurning;
      R     "MAL1S032Par".Par.FlagMachine.CmdTurnRevAfterTurning;
      R     "MAL1S032Par".Par.FlagMachine.WEGMESSUNG_0;
      R     "MAL1S032Par".Par.FlagMachine.CmdTurnFwdAfterUnloading;
      R     "MAL1S032Par".Par.FlagMachine.CmdTurnRevAfterUnloading;
      R     "MAL1S032Par".Par.FlagMachine.NULL_INDEX_FP;
//
      U     "MAL1S032".PCRead.Step.StIdling;
      O     "MAL1S032".PCRead.Step.StPassive;
      SPBN  csn;
      L     0; // clear step number
      T     "MAL1S032Par".Par.ParIntMachine.ActualStep;
      T     "MAL1S032Par".StepAct.StepNumber;
csn:  NOP   0;

NETWORK
TITLE =Main0_End: Init flag
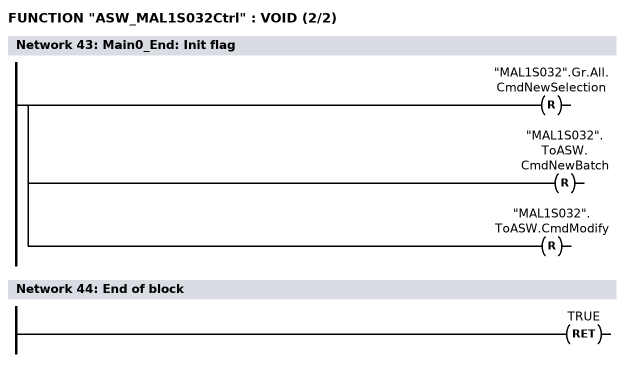

      SET   ;
      R     "MAL1S032".Gr.All.CmdNewSelection;
      R     "MAL1S032".ToASW.CmdNewBatch;
      R     "MAL1S032".ToASW.CmdModify;

NETWORK
TITLE =End of block

      BE    ;

END_FUNCTION

